Fanuc TP program (LS listing): OPN_VLE4.LS

/PROG  OPN_VLE4	  Macro
/ATTR
OWNER		= MNEDITOR;
COMMENT		= "OPEN VALVE4 (B)";
PROG_SIZE	= 522;
CREATE		= DATE 06-12-07  TIME 07:27:10;
MODIFIED	= DATE 16-07-07  TIME 08:25:50;
FILE_NAME	= ;
VERSION		= 0;
LINE_COUNT	= 13;
MEMORY_SIZE	= 850;
PROTECT		= READ;
STORAGE		= CMOS;
TCD:  STACK_SIZE	= 0,
      TASK_PRIORITY	= 50,
      TIME_SLICE	= 0,
      BUSY_LAMP_OFF	= 0,
      ABORT_REQUEST	= 0,
      PAUSE_REQUEST	= 0;
DEFAULT_GROUP	= *,*,*,*,*;
CONTROL_CODE	= 00001000 00000000;
/APPL
  HANDLING : TRUE ;
/MN
   1:  !******************************** ;
   2:  !  GM METAL FORMING GLOBAL 4 S/W ;
   3:  !******************************** ;
   4:  ! MACRO TO OPEN VALVE 4 (B POS) ;
   5:  !******************************** ;
   6:  ! 2016-04-05 Global-4 S/W Rel 4.0 ;
   7:  !******************************** ;
   8:   ;
   9:  CALL DMSTAT    ;
  10:   ;
  11:  DO[807]=OFF ;
  12:  DO[808]=ON ;
  13:   ;
/POS
/END
